// SIMATIC S7-200 project (STEP 7-Micro/WIN), CPU 221 REL 01.10

SYMBOL_TABLE USER1
start            I0.0
estop            I0.1
cb1              I0.2
cb2              I0.3
cb3              I0.4
cb4              I0.5
cb5              I0.6
cb6              I0.7
m1t              Q0.0
m1n              Q0.1
m2t              Q0.2
m2n              Q0.3
d                Q0.4
END_SYMBOL_TABLE

ORGANIZATION_BLOCK MAIN:OB1
TITLE=PROGRAM COMMENTS
BEGIN
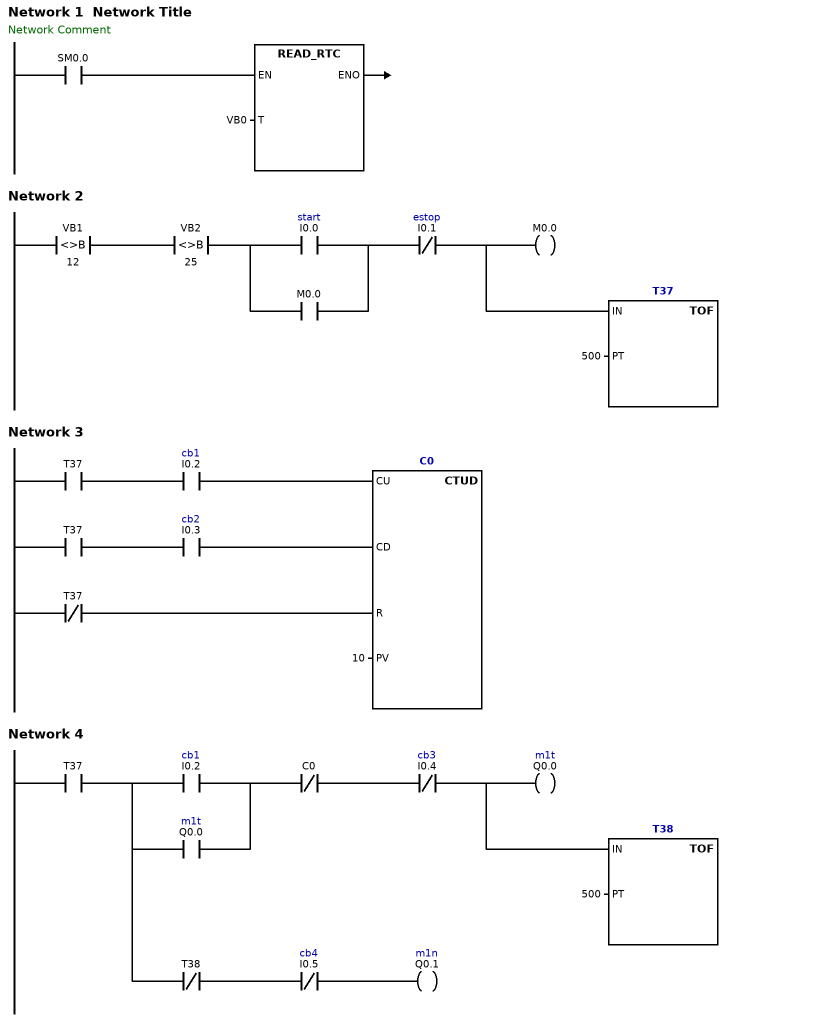
Network 1 // Network Title
// Network Comment
LD     SM0.0
TODR   VB0
Network 2
LDB<>  VB1, 12
AB<>   VB2, 25
LD     start:I0.0
O      M0.0
ALD
AN     estop:I0.1
=      M0.0
TOF    T37, 500
Network 3
LD     T37
A      cb1:I0.2
LD     T37
A      cb2:I0.3
LDN    T37
CTUD   C0, 10
Network 4
LD     T37
LPS
LD     cb1:I0.2
O      m1t:Q0.0
AN     C0
AN     cb3:I0.4
ALD
=      m1t:Q0.0
TOF    T38, 500
LPP
AN     T38
AN     cb4:I0.5
=      m1n:Q0.1
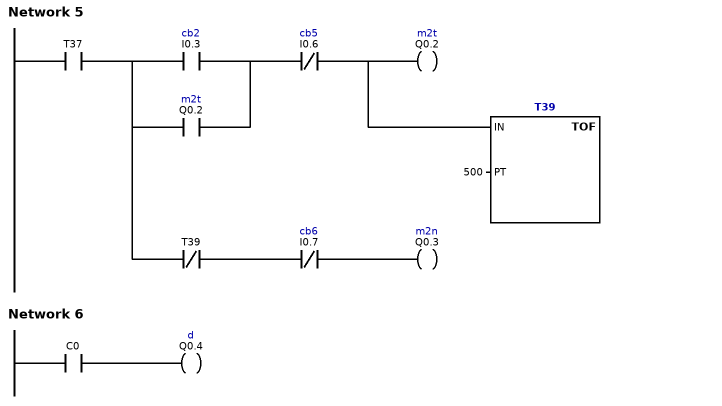
Network 5
LD     T37
LPS
LD     cb2:I0.3
O      m2t:Q0.2
AN     cb5:I0.6
ALD
=      m2t:Q0.2
TOF    T39, 500
LPP
AN     T39
AN     cb6:I0.7
=      m2n:Q0.3
Network 6
LD     C0
=      d:Q0.4
END_ORGANIZATION_BLOCK
